TYPE bsp :

UNION
	a: ARRAY[0..3] OF BYTE;
	b: DINT;
END_UNION

END_TYPE

(* stored: Version 1.1.0.1, ProductVersion 3.1.4022.16
   DUT bsp: Id {5c3398cb-77fb-4354-bfc7-ccaba91d8d65} *)
